(* CoDeSys 2.3.9.50 project: 3B.pr6 *)
(* Libraries: STANDARD.LB6 5.6.98 12:03:02 *)

(* POU MAIN, LD *)
PROGRAM MAIN
VAR
	switch AT %IX0.0: BOOL;
	t1: TON;
	FAN AT %QX0.0: BOOL;
END_VAR
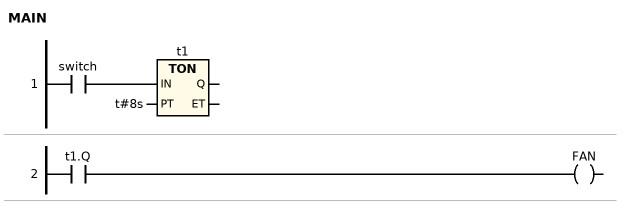
_LD_ (* Ladder Diagram *)
NETWORK 1
	[switch] - t1:TON(IN: *, PT: t#8s)
NETWORK 2
	[t1.Q] --- (FAN)
_END_LD_
(* the same logic as Structured Text *)
(* Network 1 *)
t1(IN := switch, PT := t#8s);
(* Network 2 *)
FAN := t1.Q;
END_PROGRAM
